FUNCTION_BLOCK TMIN
VAR_INPUT
	IN : BOOL;
	PT : TIME;
END_VAR
VAR_OUTPUT
	Q : BOOL;
END_VAR
VAR
	pm : TP;
END_VAR

(*
version 1.0	21. jul. 2008
programmer 	hugo
tested by	oscat

Q of tMIN will follow IN except that it forces a minimum ontime for the output Q.

*)

pm(in := IN, PT := PT);
Q := IN OR pm.Q;


(* revision history
hm	21. jul. 2008	rev 1.0
	original version

*)

END_FUNCTION_BLOCK

(* stored: Version 1.1.0.1, ProductVersion 3.1.4022.7
   POU TMIN: Id {15afba2d-6c59-42d4-bcd3-f8cc94b444cc}, SpecialFunc None *)
